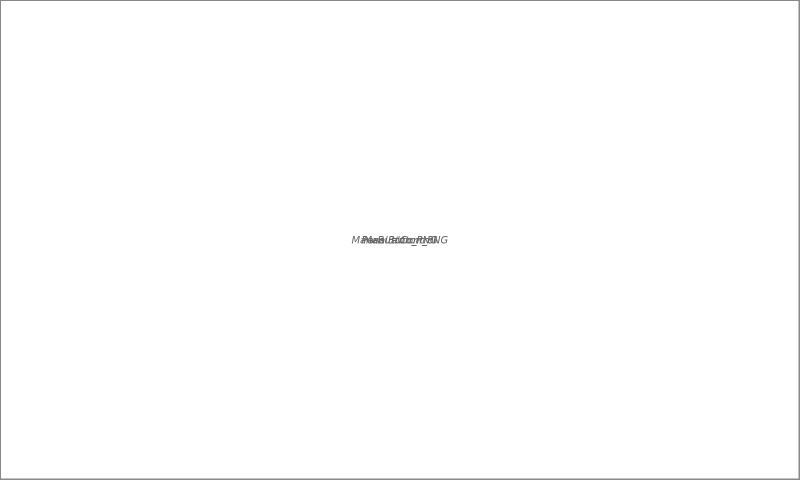
VISUALIZATION Manual_PNG  // 800x480
VAR_IN_OUT
	bCmdManual  	: BOOL ; // switch to manual screen
	bCmdParameter	: BOOL ; // switch to parameter screen
END_VAR
    Frame (0,0 800x480)
        shows ManualButton_PNG(bCmdManual := bCmdManual)
    Frame (0,0 800x480)
        shows ManualControl()
    Frame (0,0 800x480)
        shows ParButton_PNG(bCmdParameter := bCmdParameter)
END_VISUALIZATION

(* stored: Version 1.1.0.1, ProductVersion 3.1.4024.5
   Visu Manual_PNG: Id {6ebf1ffe-3d8a-4c3c-ace5-8874cf269357} *)
